PROGRAM prgComEffIO
VAR
	fbCom		: FB_MqttCommunicator_V2;
	f_Trig_HB: f_trig;
	stringArray_Last_HB: ARRAY[0..50] OF STRING(30);
	intCount: INT;
	time_Temp: TIME;
	time_HB: TIME:= T#15S;
END_VAR

fbCom(
	bConnect:= TRUE, 
	sUserName:= 'b472a324-06e3-4d07-96cf-574b1847d8ff', 
	sUserPassword:= '5b687dd8-7c3c-4e3c-8272-e8ed6dc08177', 
	strAuthKey:= 'EIO08031879806', 
	eSavePositionCertificate:= eSavePositionOnPLC.ePostionHardDisk, 
	time_HeartBeat_sec := time_HB,
	bConnected=> , 
	bError=> , 
	hrErrorCode=> , 
	eConnectionState=> , 
	eErrorMessage_Out=> );
	
f_Trig_HB(CLK :=  fbCom.bHBSending);



prg_SystemTime();

IF f_Trig_HB.Q THEN
	stringArray_Last_HB[intCount] := prg_SystemTime.stringSystemTime_ms;
	intCount := intCount+1;
	IF intCount>50 OR intCount<0 THEN
		intCount:=0;
	END_IF
	stringArray_Last_HB[intCount] := '';
END_IF

time_Temp := fbCom.fbTimerHB.ET;

END_PROGRAM

(* stored: Version 1.1.0.1, ProductVersion 3.1.4024.12
   POU prgComEffIO: Id {cbcd318b-bf51-484c-bcaa-d6efcdf43fe3}, SpecialFunc None *)
